KUKA KRL program: dai_sen_validation_01.src, dai_sen_validation_01.dat

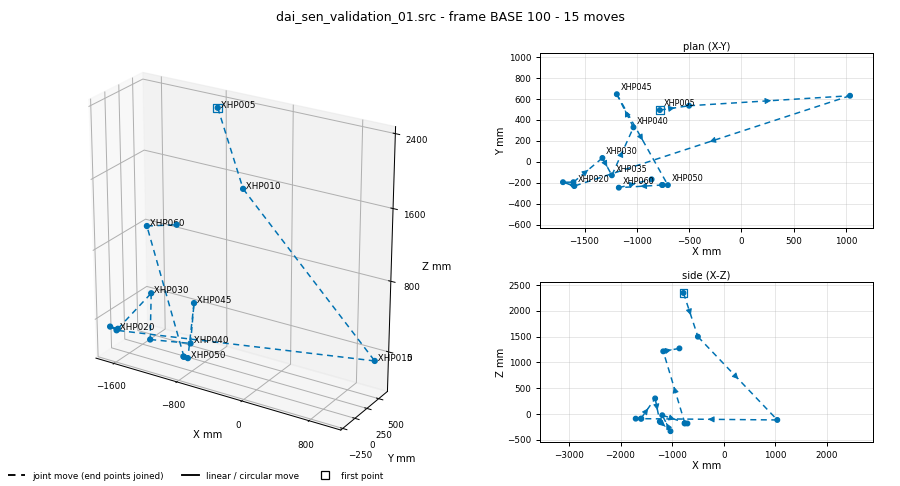
[picture p0: tool path of dai_sen_validation_01.src in frame BASE 100, 15 of 17 moves have a stored position in this frame; points joined in program order, loops and branches not executed]
--- dai_sen_validation_01.src ---
&ACCESS RVP
&REL 21
&PARAM DISKPATH = KRC:\R1\H_Prog
DEF dai_sen_validation_01( )
;FOLD INI;%{PE}
  ;FOLD BASISTECH INI
    GLOBAL INTERRUPT DECL 3 WHEN $STOPMESS==TRUE DO IR_STOPM ( )
    INTERRUPT ON 3
    BAS (#INITMOV,0 )
  ;ENDFOLD (BASISTECH INI)
  ;FOLD USER INI
    ;Make your modifications here
  ;ENDFOLD (USER INI)
;ENDFOLD (INI)
;FOLD ; Anlagenbezeichn: HC51_C    Stations-Nr: 080RB_100;%{PE}
;FOLD Parameters ;%{h}
;Params IlfProvider=kukaroboter.basistech.inlineforms.comments.comment; Kuka.Content=Anlagenbezeichn: HC51_C    Stations-Nr: 080RB_100
;ENDFOLD
;ENDFOLD
;FOLD ; Stand / Version: V1.0;%{PE}
;FOLD Parameters ;%{h}
;Params IlfProvider=kukaroboter.basistech.inlineforms.comments.comment; Kuka.Content=Stand / Version: V1.0
;ENDFOLD
;ENDFOLD
;FOLD ; Name Bearbeiter: EBZ-AE;%{PE}
;FOLD Parameters ;%{h}
;Params IlfProvider=kukaroboter.basistech.inlineforms.comments.comment; Kuka.Content=Name Bearbeiter: EBZ-AE
;ENDFOLD
;ENDFOLD
;FOLD ; Translator Version:29.01.2024 - Version 15.08;%{PE}
;FOLD Parameters ;%{h}
;Params IlfProvider=kukaroboter.basistech.inlineforms.comments.comment; Kuka.Content=Translator Version:29.01.2024 - Version 15.08
;ENDFOLD
;ENDFOLD


;FOLD ; This program has been cleaned by KANERT_Makro. High risk of crash!!! Check the program carefully before deleting this comment. ;%{PE}
;FOLD Parameters ;%{h}
;Params IlfProvider=kukaroboter.basistech.inlineforms.comments.comment; Kuka.Content=This program has been cleaned by KANERT_Makro. High risk of crash!!! Check the program carefully before deleting this comment.
;ENDFOLD
WAIT FOR FALSE
;ENDFOLD
;check program once again after mounting calibration plate
WAIT FOR FALSE ;STATUS
;PROGRAM CHECKED BY: Szala
;COLLISIONS NOT CHECKED
;FOLD PTP HOME Vel=100 % DEFAULT;%{PE}
;FOLD Parameters ;%{h}
;Params IlfProvider=kukaroboter.basistech.inlineforms.movement.old; Kuka.IsGlobalPoint=False; Kuka.PointName=HOME; Kuka.BlendingEnabled=False; Kuka.MoveDataPtpName=DEFAULT; Kuka.VelocityPtp=100; Kuka.CurrentCDSetIndex=0; Kuka.MovementParameterFieldEnabled=True; IlfCommand=PTP
;ENDFOLD
$BWDSTART = FALSE
PDAT_ACT = PDEFAULT
FDAT_ACT = FHOME
BAS(#PTP_PARAMS, 100.0)
SET_CD_PARAMS (0)
PTP XHOME
;ENDFOLD

;Dynamische Pruefung Teil vorhanden
;FOLD PartPresent.CheckOff #1:5279, #2:5280, #3:1025, #4:1025, #5:1025, #6:1025, Bounce Time:100, Constant: Yes;%{PE}%
CheckPartPresent(5279,5280,1025,1025,1025,1025,100, True,FALSE)
;ENDFOLD

;Greifer-Ventile betatigen/pruefen
;FOLD DAI_GripValveCheck.Valve2 State:Fixierstift Ausfahren Gs, 080GRH101-QM1;%{PE}%
CheckValveState(2,1)
;ENDFOLD
;FOLD DAI_GripValveCheck.Valve3 State:Spanner Oeffnen Gs, 080GRH101-QM2;%{PE}%
CheckValveState(3,1)
;ENDFOLD
;FOLD DAI_GripValveCheck.Valve4 State:Sauger Abblasen Gs, 080GRH101-QM3;%{PE}%
CheckValveState(4,1)
;ENDFOLD
;FOLD DAI_GripValveCheck.Valve5 State:Sauger Abblasen Gs, 080GRH101-QM4;%{PE}%
CheckValveState(5,1)
;ENDFOLD

;Camera Initialisieren und Docken
;
;FOLD DAI_SEN.INIT Nbr of cams:1;%{PE}%
; SEN_MaxCams=1
; DAI_SEN_CMD ( #INIT )
;;ENDFOLD

;
;
;FOLD DAI_SEN.CHANGEJOB Cam:1, Job nbr.:1;%{PE}%
; SEN_Cam=1
; DAI_SEN_CMD ( #ChangeJob )
;;ENDFOLD

;FOLD PTP HP005 CONT Vel=100 % PDAT1 Tool[110]:MSK_01_XYa_Sensopart Base[100]:SENSOPART_CALIBRATEPLATE ;%{PE}
;FOLD Parameters ;%{h}
;Params IlfProvider=kukaroboter.basistech.inlineforms.movement.old; Kuka.IsGlobalPoint=False; Kuka.PointName=HP005; Kuka.BlendingEnabled=True; Kuka.MoveDataPtpName=PDAT1; Kuka.VelocityPtp=100; Kuka.CurrentCDSetIndex=0; Kuka.MovementParameterFieldEnabled=True; IlfCommand=PTP
;ENDFOLD
$BWDSTART = FALSE
PDAT_ACT = PPDAT1
FDAT_ACT = FHP005
BAS(#PTP_PARAMS, 100.0)
SET_CD_PARAMS (0)
PTP XHP005 C_Dis
;ENDFOLD
;FOLD PTP HP010 CONT Vel=100 % PDAT2 Tool[110]:MSK_01_XYa_Sensopart Base[100]:SENSOPART_CALIBRATEPLATE ;%{PE}
;FOLD Parameters ;%{h}
;Params IlfProvider=kukaroboter.basistech.inlineforms.movement.old; Kuka.IsGlobalPoint=False; Kuka.PointName=HP010; Kuka.BlendingEnabled=True; Kuka.MoveDataPtpName=PDAT2; Kuka.VelocityPtp=100; Kuka.CurrentCDSetIndex=0; Kuka.MovementParameterFieldEnabled=True; IlfCommand=PTP
;ENDFOLD
$BWDSTART = FALSE
PDAT_ACT = PPDAT2
FDAT_ACT = FHP010
BAS(#PTP_PARAMS, 100.0)
SET_CD_PARAMS (0)
PTP XHP010 C_Dis
;ENDFOLD
;FOLD PTP HP015 CONT Vel=100 % PDAT3 Tool[110]:MSK_01_XYa_Sensopart Base[100]:SENSOPART_CALIBRATEPLATE ;%{PE}
;FOLD Parameters ;%{h}
;Params IlfProvider=kukaroboter.basistech.inlineforms.movement.old; Kuka.IsGlobalPoint=False; Kuka.PointName=HP015; Kuka.BlendingEnabled=True; Kuka.MoveDataPtpName=PDAT3; Kuka.VelocityPtp=100; Kuka.CurrentCDSetIndex=0; Kuka.MovementParameterFieldEnabled=True; IlfCommand=PTP
;ENDFOLD
$BWDSTART = FALSE
PDAT_ACT = PPDAT3
FDAT_ACT = FHP015
BAS(#PTP_PARAMS, 100.0)
SET_CD_PARAMS (0)
PTP XHP015 C_Dis
;ENDFOLD
;FOLD PTP HP020 Vel=100 % PDAT4 Tool[110]:MSK_01_XYa_Sensopart Base[100]:SENSOPART_CALIBRATEPLATE ;%{PE}
;FOLD Parameters ;%{h}
;Params IlfProvider=kukaroboter.basistech.inlineforms.movement.old; Kuka.IsGlobalPoint=False; Kuka.PointName=HP020; Kuka.BlendingEnabled=False; Kuka.MoveDataPtpName=PDAT4; Kuka.VelocityPtp=100; Kuka.CurrentCDSetIndex=0; Kuka.MovementParameterFieldEnabled=True; IlfCommand=PTP
;ENDFOLD
$BWDSTART = FALSE
PDAT_ACT = PPDAT4
FDAT_ACT = FHP020
BAS(#PTP_PARAMS, 100.0)
SET_CD_PARAMS (0)
PTP XHP020
;ENDFOLD
;FOLD LIN SEN520W080_005 Vel=0.2 m/s CPDAT5 Tool[110]:MSK_01_XYa_Sensopart Base[100]:SENSOPART_CALIBRATEPLATE ;%{PE}
;FOLD Parameters ;%{h}
;Params IlfProvider=kukaroboter.basistech.inlineforms.movement.old; Kuka.IsGlobalPoint=False; Kuka.PointName=SEN520W080_005; Kuka.BlendingEnabled=False; Kuka.MoveDataName=CPDAT5; Kuka.VelocityPath=0.2; Kuka.CurrentCDSetIndex=0; Kuka.MovementParameterFieldEnabled=True; IlfCommand=LIN
;ENDFOLD
$BWDSTART = FALSE
LDAT_ACT = LCPDAT5
FDAT_ACT = FSEN520W080_005
BAS(#CP_PARAMS, 0.2)
SET_CD_PARAMS (0)
LIN XSEN520W080_005
;ENDFOLD

;
;FOLD DAI_SEN.VALIDATION Waiting Time: 0 s, Job nbr.: 1, Cam: 1, Calibration Base/Tool: 110 ;%{PE}
; SEN_CalibMode=1
; SEN_JobResponse=1
; SEN_TimeOut=0
; SEN_CalibBase=110
; SEN_Cam=1
; DAI_SEN_CMD ( #CALIBRATION )
;;ENDFOLD

;Kalibrationposition
;Fokus-Abstand Kamera zur Kalibrierplatte 170mm

;
;FOLD DAI_SEN.CHANGEJOB Cam: 1, Job nbr.: 1 ;%{PE}
; SEN_Cam=1
; SEN_JobResponse=1
; DAI_SEN_CMD ( #ChangeJob )
;;ENDFOLD

;
;FOLD DAI_SEN.CALIBRATION Cam: 1, Calibration Base/Tool: 30, Waiting Time: 1 s ;%{PE}
; SEN_CalibMode=2
; SEN_JobResponse=1
; SEN_TimeOut=1
; SEN_CalibBase=30
; SEN_Cam=1
; SEN_CopyMode=1
; DAI_SEN_CMD ( #CALIBRATION )
;;ENDFOLD

;FOLD LIN HP025 Vel=0.2 m/s CPDAT6 Tool[110]:MSK_01_XYa_Sensopart Base[100]:SENSOPART_CALIBRATEPLATE ;%{PE}
;FOLD Parameters ;%{h}
;Params IlfProvider=kukaroboter.basistech.inlineforms.movement.old; Kuka.IsGlobalPoint=False; Kuka.PointName=HP025; Kuka.BlendingEnabled=False; Kuka.MoveDataName=CPDAT6; Kuka.VelocityPath=0.2; Kuka.CurrentCDSetIndex=0; Kuka.MovementParameterFieldEnabled=True; IlfCommand=LIN
;ENDFOLD
$BWDSTART = FALSE
LDAT_ACT = LCPDAT6
FDAT_ACT = FHP025
BAS(#CP_PARAMS, 0.2)
SET_CD_PARAMS (0)
LIN XHP025
;ENDFOLD
;FOLD PTP HP030 CONT Vel=100 % PDAT7 Tool[110]:MSK_01_XYa_Sensopart Base[100]:SENSOPART_CALIBRATEPLATE ;%{PE}
;FOLD Parameters ;%{h}
;Params IlfProvider=kukaroboter.basistech.inlineforms.movement.old; Kuka.IsGlobalPoint=False; Kuka.PointName=HP030; Kuka.BlendingEnabled=True; Kuka.MoveDataPtpName=PDAT7; Kuka.VelocityPtp=100; Kuka.CurrentCDSetIndex=0; Kuka.MovementParameterFieldEnabled=True; IlfCommand=PTP
;ENDFOLD
$BWDSTART = FALSE
PDAT_ACT = PPDAT7
FDAT_ACT = FHP030
BAS(#PTP_PARAMS, 100.0)
SET_CD_PARAMS (0)
PTP XHP030 C_Dis
;ENDFOLD
;FOLD PTP HP035 CONT Vel=100 % PDAT8 Tool[110]:MSK_01_XYa_Sensopart Base[100]:SENSOPART_CALIBRATEPLATE ;%{PE}
;FOLD Parameters ;%{h}
;Params IlfProvider=kukaroboter.basistech.inlineforms.movement.old; Kuka.IsGlobalPoint=False; Kuka.PointName=HP035; Kuka.BlendingEnabled=True; Kuka.MoveDataPtpName=PDAT8; Kuka.VelocityPtp=100; Kuka.CurrentCDSetIndex=0; Kuka.MovementParameterFieldEnabled=True; IlfCommand=PTP
;ENDFOLD
$BWDSTART = FALSE
PDAT_ACT = PPDAT8
FDAT_ACT = FHP035
BAS(#PTP_PARAMS, 100.0)
SET_CD_PARAMS (0)
PTP XHP035 C_Dis
;ENDFOLD
;FOLD PTP HP040 CONT Vel=100 % PDAT9 Tool[111]:MSK_02_XYa_Sensopart Base[100]:SENSOPART_CALIBRATEPLATE ;%{PE}
;FOLD Parameters ;%{h}
;Params IlfProvider=kukaroboter.basistech.inlineforms.movement.old; Kuka.IsGlobalPoint=False; Kuka.PointName=HP040; Kuka.BlendingEnabled=True; Kuka.MoveDataPtpName=PDAT9; Kuka.VelocityPtp=100; Kuka.CurrentCDSetIndex=0; Kuka.MovementParameterFieldEnabled=True; IlfCommand=PTP
;ENDFOLD
$BWDSTART = FALSE
PDAT_ACT = PPDAT9
FDAT_ACT = FHP040
BAS(#PTP_PARAMS, 100.0)
SET_CD_PARAMS (0)
PTP XHP040 C_Dis
;ENDFOLD
;FOLD PTP HP045 CONT Vel=100 % PDAT10 Tool[111]:MSK_02_XYa_Sensopart Base[100]:SENSOPART_CALIBRATEPLATE ;%{PE}
;FOLD Parameters ;%{h}
;Params IlfProvider=kukaroboter.basistech.inlineforms.movement.old; Kuka.IsGlobalPoint=False; Kuka.PointName=HP045; Kuka.BlendingEnabled=True; Kuka.MoveDataPtpName=PDAT10; Kuka.VelocityPtp=100; Kuka.CurrentCDSetIndex=0; Kuka.MovementParameterFieldEnabled=True; IlfCommand=PTP
;ENDFOLD
$BWDSTART = FALSE
PDAT_ACT = PPDAT10
FDAT_ACT = FHP045
BAS(#PTP_PARAMS, 100.0)
SET_CD_PARAMS (0)
PTP XHP045 C_Dis
;ENDFOLD
;FOLD PTP HP050 Vel=100 % PDAT11 Tool[111]:MSK_02_XYa_Sensopart Base[100]:SENSOPART_CALIBRATEPLATE ;%{PE}
;FOLD Parameters ;%{h}
;Params IlfProvider=kukaroboter.basistech.inlineforms.movement.old; Kuka.IsGlobalPoint=False; Kuka.PointName=HP050; Kuka.BlendingEnabled=False; Kuka.MoveDataPtpName=PDAT11; Kuka.VelocityPtp=100; Kuka.CurrentCDSetIndex=0; Kuka.MovementParameterFieldEnabled=True; IlfCommand=PTP
;ENDFOLD
$BWDSTART = FALSE
PDAT_ACT = PPDAT11
FDAT_ACT = FHP050
BAS(#PTP_PARAMS, 100.0)
SET_CD_PARAMS (0)
PTP XHP050
;ENDFOLD
;FOLD LIN SEN520W080_010 Vel=0.2 m/s CPDAT12 Tool[111]:MSK_02_XYa_Sensopart Base[100]:SENSOPART_CALIBRATEPLATE ;%{PE}
;FOLD Parameters ;%{h}
;Params IlfProvider=kukaroboter.basistech.inlineforms.movement.old; Kuka.IsGlobalPoint=False; Kuka.PointName=SEN520W080_010; Kuka.BlendingEnabled=False; Kuka.MoveDataName=CPDAT12; Kuka.VelocityPath=0.2; Kuka.CurrentCDSetIndex=0; Kuka.MovementParameterFieldEnabled=True; IlfCommand=LIN
;ENDFOLD
$BWDSTART = FALSE
LDAT_ACT = LCPDAT12
FDAT_ACT = FSEN520W080_010
BAS(#CP_PARAMS, 0.2)
SET_CD_PARAMS (0)
LIN XSEN520W080_010
;ENDFOLD

;
;FOLD DAI_SEN.VALIDATION Waiting Time: 0 s, Job nbr.: 1, Cam: 1, Calibration Base/Tool: 110 ;%{PE}
; SEN_CalibMode=1
; SEN_JobResponse=1
; SEN_TimeOut=0
; SEN_CalibBase=110
; SEN_Cam=1
; DAI_SEN_CMD ( #CALIBRATION )
;;ENDFOLD

;Kalibrationposition
;Fokus-Abstand Kamera zur Kalibrierplatte 170mm

;
;FOLD DAI_SEN.CHANGEJOB Cam: 1, Job nbr.: 1 ;%{PE}
; SEN_Cam=1
; SEN_JobResponse=1
; DAI_SEN_CMD ( #ChangeJob )
;;ENDFOLD

;
;FOLD DAI_SEN.CALIBRATION Cam: 1, Calibration Base/Tool: 30, Waiting Time: 1 s ;%{PE}
; SEN_CalibMode=2
; SEN_JobResponse=1
; SEN_TimeOut=1
; SEN_CalibBase=30
; SEN_Cam=1
; SEN_CopyMode=1
; DAI_SEN_CMD ( #CALIBRATION )
;;ENDFOLD

;FOLD LIN HP055 Vel=0.2 m/s CPDAT13 Tool[111]:MSK_02_XYa_Sensopart Base[100]:SENSOPART_CALIBRATEPLATE ;%{PE}
;FOLD Parameters ;%{h}
;Params IlfProvider=kukaroboter.basistech.inlineforms.movement.old; Kuka.IsGlobalPoint=False; Kuka.PointName=HP055; Kuka.BlendingEnabled=False; Kuka.MoveDataName=CPDAT13; Kuka.VelocityPath=0.2; Kuka.CurrentCDSetIndex=0; Kuka.MovementParameterFieldEnabled=True; IlfCommand=LIN
;ENDFOLD
$BWDSTART = FALSE
LDAT_ACT = LCPDAT13
FDAT_ACT = FHP055
BAS(#CP_PARAMS, 0.2)
SET_CD_PARAMS (0)
LIN XHP055
;ENDFOLD
;FOLD PTP HP060 CONT Vel=100 % PDAT14 Tool[111]:MSK_02_XYa_Sensopart Base[100]:SENSOPART_CALIBRATEPLATE ;%{PE}
;FOLD Parameters ;%{h}
;Params IlfProvider=kukaroboter.basistech.inlineforms.movement.old; Kuka.IsGlobalPoint=False; Kuka.PointName=HP060; Kuka.BlendingEnabled=True; Kuka.MoveDataPtpName=PDAT14; Kuka.VelocityPtp=100; Kuka.CurrentCDSetIndex=0; Kuka.MovementParameterFieldEnabled=True; IlfCommand=PTP
;ENDFOLD
$BWDSTART = FALSE
PDAT_ACT = PPDAT14
FDAT_ACT = FHP060
BAS(#PTP_PARAMS, 100.0)
SET_CD_PARAMS (0)
PTP XHP060 C_Dis
;ENDFOLD
;FOLD PTP HP065 CONT Vel=100 % PDAT15 Tool[111]:MSK_02_XYa_Sensopart Base[100]:SENSOPART_CALIBRATEPLATE ;%{PE}
;FOLD Parameters ;%{h}
;Params IlfProvider=kukaroboter.basistech.inlineforms.movement.old; Kuka.IsGlobalPoint=False; Kuka.PointName=HP065; Kuka.BlendingEnabled=True; Kuka.MoveDataPtpName=PDAT15; Kuka.VelocityPtp=100; Kuka.CurrentCDSetIndex=0; Kuka.MovementParameterFieldEnabled=True; IlfCommand=PTP
;ENDFOLD
$BWDSTART = FALSE
PDAT_ACT = PPDAT15
FDAT_ACT = FHP065
BAS(#PTP_PARAMS, 100.0)
SET_CD_PARAMS (0)
PTP XHP065 C_Dis
;ENDFOLD

;FOLD PTP HOME Vel=100 % DEFAULT;%{PE}
;FOLD Parameters ;%{h}
;Params IlfProvider=kukaroboter.basistech.inlineforms.movement.old; Kuka.IsGlobalPoint=False; Kuka.PointName=HOME; Kuka.BlendingEnabled=False; Kuka.MoveDataPtpName=DEFAULT; Kuka.VelocityPtp=100; Kuka.CurrentCDSetIndex=0; Kuka.MovementParameterFieldEnabled=True; IlfCommand=PTP
;ENDFOLD
$BWDSTART = FALSE
PDAT_ACT = PDEFAULT
FDAT_ACT = FHOME
BAS(#PTP_PARAMS, 100.0)
SET_CD_PARAMS (0)
PTP XHOME
;ENDFOLD

END

--- dai_sen_validation_01.dat ---
&ACCESS  RVP
&REL 5

DEFDAT  DAI_SEN_VALIDATION_01
DECL MODULEPARAM_T LAST_TP_PARAMS={PARAMS[] "Kuka.PointName=HP006; Kuka.FrameData.base_no=100; Kuka.FrameData.tool_no=110; Kuka.FrameData.ipo_frame=#BASE; Kuka.FrameData.point2=; Kuka.isglobalpoint=False; Kuka.MoveDataPtpName=PDAT4; Kuka.MovementDataPdat.apo_mode=#CDIS; Kuka.MovementDataPdat.apo_dist=0; Kuka.MovementData.vel=100; Kuka.MovementData.acc=100; Kuka.MovementData.exax_ign=0; Kuka.VelocityPtp=100; Kuka.BlendingEnabled=True; Kuka.APXEnabled=False; Kuka.CurrentCDSetIndex=0 "}

; E6POS Declarations
DECL E6POS XHP005={X -779.682373,Y 494.501343,Z 2348.19165,A -175.757172,B 17.4713459,C 131.541290,S 18,T 43,E1 -2600.00,E2 0.0,E3 0.0,E4 0.0,E5 0.0,E6 0.0}
DECL E6POS XHP010={X -500.096771,Y 536.086365,Z 1500.18787,A -169.213486,B 34.4074,C 149.267181,S 18,T 43,E1 -2600.00,E2 0.0,E3 0.0,E4 0.0,E5 0.0,E6 0.0}
DECL E6POS XHP015={X 1039.36145,Y 631.731934,Z -114.176437,A -93.1385803,B 54.9452362,C -88.7430191,S 18,T 43,E1 -2600.00,E2 0.0,E3 0.0,E4 0.0,E5 0.0,E6 0.0}
DECL E6POS XHP020={X -1596.92188,Y -231.733139,Z -89.1872864,A -89.0549,B 40.0358,C -90.0032425,S 18,T 43,E1 -205.766190,E2 0.0,E3 0.0,E4 0.0,E5 0.0,E6 0.0}
DECL E6POS XSEN520W080_005={X -1705.99988,Y -194.989441,Z -89.0150375,A -89.9998856,B 40.0002289,C -89.9999084,S 18,T 43,E1 -200.000,E2 0.0,E3 0.0,E4 0.0,E5 0.0,E6 0.0}
DECL E6POS XHP025={X -1606.01245,Y -194.991440,Z -89.0240707,A -89.9998856,B 40.0002289,C -89.9999161,S 18,T 43,E1 -200.000,E2 0.0,E3 0.0,E4 0.0,E5 0.0,E6 0.0}
DECL E6POS XHP030={X -1328.80969,Y 36.5054893,Z 303.534821,A -152.227,B 60.2150650,C 96.8617401,S 18,T 43,E1 -1655.49500,E2 0.0,E3 0.0,E4 0.0,E5 0.0,E6 0.0}
DECL E6POS XHP035={X -1238.37817,Y -129.287674,Z -146.624466,A -106.527870,B 71.9081802,C 131.198608,S 18,T 43,E1 -1655.50,E2 0.0,E3 0.0,E4 0.0,E5 0.0,E6 0.0}
DECL E6POS XHP040={X -1031.76807,Y 329.438507,Z -332.201782,A -93.8291092,B 73.7938156,C 125.149490,S 18,T 43,E1 -1655.50,E2 0.0,E3 0.0,E4 0.0,E5 0.0,E6 0.0}
DECL E6POS XHP045={X -1190.97339,Y 646.372437,Z -22.7895660,A -163.509048,B 67.4667282,C 23.6408825,S 18,T 11,E1 -1655.50,E2 0.0,E3 0.0,E4 0.0,E5 0.0,E6 0.0}
DECL E6POS XHP050={X -702.601318,Y -223.040100,Z -182.489,A 93.7801285,B 64.4597321,C 95.9688339,S 18,T 3,E1 -1804.39478,E2 0.0,E3 0.0,E4 0.0,E5 0.0,E6 0.0}
DECL E6POS XSEN520W080_010={X -758.815063,Y -221.481491,Z -179.966537,A 93.7779083,B 64.4604187,C 95.9661331,S 18,T 3,E1 -1804.39478,E2 0.0,E3 0.0,E4 0.0,E5 0.0,E6 0.0}
DECL E6POS XHP055={X -751.930664,Y -221.674210,Z -180.276016,A 93.7779083,B 64.4604187,C 95.9661331,S 18,T 3,E1 -1804.39478,E2 0.0,E3 0.0,E4 0.0,E5 0.0,E6 0.0}
DECL E6POS XHP060={X -1171.94519,Y -247.431534,Z 1216.17859,A 177.204590,B 36.6070137,C -34.5379028,S 18,T 3,E1 -2533.72266,E2 0.0,E3 0.0,E4 0.0,E5 0.0,E6 0.0}
DECL E6POS XHP065={X -858.226135,Y -167.701263,Z 1273.28308,A 176.900,B 34.6558075,C -12.6554432,S 18,T 35,E1 -2620.65845,E2 0.0,E3 0.0,E4 0.0,E5 0.0,E6 0.0}

; PDAT/LDAT Declarations
DECL PDAT PPDAT1={VEL 100.000,ACC 100.000,APO_DIST 0.0,APO_MODE #CDIS,GEAR_JERK 50.0000,EXAX_IGN 0}
DECL PDAT PPDAT2={VEL 100.000,ACC 100.000,APO_DIST 0.0,APO_MODE #CDIS,GEAR_JERK 50.0000,EXAX_IGN 0}
DECL PDAT PPDAT3={VEL 100.000,ACC 100.000,APO_DIST 0.0,APO_MODE #CDIS,GEAR_JERK 50.0000,EXAX_IGN 0}
DECL PDAT PPDAT4={VEL 100.000,ACC 100.000,APO_DIST 0.0,APO_MODE #CDIS,GEAR_JERK 50.0000,EXAX_IGN 0}
DECL LDAT LCPDAT5={VEL 0.200000,ACC 100.000,APO_DIST 0.0,APO_FAC 50.0000,AXIS_VEL 100.000,AXIS_ACC 100.000,ORI_TYP #VAR,CIRC_TYP #BASE,JERK_FAC 50.0000,GEAR_JERK 50.0000,EXAX_IGN 0}
DECL LDAT LCPDAT6={VEL 0.200000,ACC 100.000,APO_DIST 0.0,APO_FAC 50.0000,AXIS_VEL 100.000,AXIS_ACC 100.000,ORI_TYP #VAR,CIRC_TYP #BASE,JERK_FAC 50.0000,GEAR_JERK 50.0000,EXAX_IGN 0}
DECL PDAT PPDAT7={VEL 100.000,ACC 100.000,APO_DIST 0.0,APO_MODE #CDIS,GEAR_JERK 50.0000,EXAX_IGN 0}
DECL PDAT PPDAT8={VEL 100.000,ACC 100.000,APO_DIST 0.0,APO_MODE #CDIS,GEAR_JERK 50.0000,EXAX_IGN 0}
DECL PDAT PPDAT9={VEL 100.000,ACC 100.000,APO_DIST 0.0,APO_MODE #CDIS,GEAR_JERK 50.0000,EXAX_IGN 0}
DECL PDAT PPDAT10={VEL 100.000,ACC 100.000,APO_DIST 0.0,APO_MODE #CDIS,GEAR_JERK 50.0000,EXAX_IGN 0}
DECL PDAT PPDAT11={VEL 100.000,ACC 100.000,APO_DIST 0.0,APO_MODE #CDIS,GEAR_JERK 50.0000,EXAX_IGN 0}
DECL LDAT LCPDAT12={VEL 0.200000,ACC 100.000,APO_DIST 0.0,APO_FAC 50.0000,AXIS_VEL 100.000,AXIS_ACC 100.000,ORI_TYP #VAR,CIRC_TYP #BASE,JERK_FAC 50.0000,GEAR_JERK 50.0000,EXAX_IGN 0}
DECL LDAT LCPDAT13={VEL 0.200000,ACC 100.000,APO_DIST 0.0,APO_FAC 50.0000,AXIS_VEL 100.000,AXIS_ACC 100.000,ORI_TYP #VAR,CIRC_TYP #BASE,JERK_FAC 50.0000,GEAR_JERK 50.0000,EXAX_IGN 0}
DECL PDAT PPDAT14={VEL 100.000,ACC 100.000,APO_DIST 0.0,APO_MODE #CDIS,GEAR_JERK 50.0000,EXAX_IGN 0}
DECL PDAT PPDAT15={VEL 100.000,ACC 100.000,APO_DIST 0.0,APO_MODE #CDIS,GEAR_JERK 50.0000,EXAX_IGN 0}

; FDAT Declarations
DECL FDAT FHOME={TOOL_NO 110,BASE_NO 100,IPO_FRAME #BASE,POINT2[] " "}
DECL FDAT FHP005={TOOL_NO 110,BASE_NO 100,IPO_FRAME #BASE,POINT2[] " "}
DECL FDAT FHP010={TOOL_NO 110,BASE_NO 100,IPO_FRAME #BASE,POINT2[] " "}
DECL FDAT FHP015={TOOL_NO 110,BASE_NO 100,IPO_FRAME #BASE,POINT2[] " "}
DECL FDAT FHP020={TOOL_NO 110,BASE_NO 100,IPO_FRAME #BASE,POINT2[] " "}
DECL FDAT FSEN520W080_005={TOOL_NO 110,BASE_NO 100,IPO_FRAME #BASE,POINT2[] " "}
DECL FDAT FHP025={TOOL_NO 110,BASE_NO 100,IPO_FRAME #BASE,POINT2[] " "}
DECL FDAT FHP030={TOOL_NO 110,BASE_NO 100,IPO_FRAME #BASE,POINT2[] " "}
DECL FDAT FHP035={TOOL_NO 110,BASE_NO 100,IPO_FRAME #BASE,POINT2[] " "}
DECL FDAT FHP040={TOOL_NO 111,BASE_NO 100,IPO_FRAME #BASE,POINT2[] " "}
DECL FDAT FHP045={TOOL_NO 111,BASE_NO 100,IPO_FRAME #BASE,POINT2[] " "}
DECL FDAT FHP050={TOOL_NO 111,BASE_NO 100,IPO_FRAME #BASE,POINT2[] " "}
DECL FDAT FSEN520W080_010={TOOL_NO 111,BASE_NO 100,IPO_FRAME #BASE,POINT2[] " "}
DECL FDAT FHP055={TOOL_NO 111,BASE_NO 100,IPO_FRAME #BASE,POINT2[] " "}
DECL FDAT FHP060={TOOL_NO 111,BASE_NO 100,IPO_FRAME #BASE,POINT2[] " "}
DECL FDAT FHP065={TOOL_NO 111,BASE_NO 100,IPO_FRAME #BASE,POINT2[] " "}

ENDDAT
